FUNCTION_BLOCK FB_Servo
VAR_INPUT
	CAMTABLE		: MC_CAM_REF;
END_VAR
VAR_OUTPUT
END_VAR
VAR
	McPower: MC_Power;
	McReset: MC_Reset;
	McMoveAbs: MC_MoveAbsolute;
	McCamIN: MC_CamIn_V2;
	McCamOUT: MC_CamOut;
	McStop: MC_Stop;
	McWrite: MC_WriteMotionFunction;
	McRead: MC_ReadMotionFunction;
END_VAR
VAR_IN_OUT
	Axis			:	AXIS_REF;
	Slave			:	AXIS_REf;
	stAxisInterface	:	ST_AxisInterface;
END_VAR

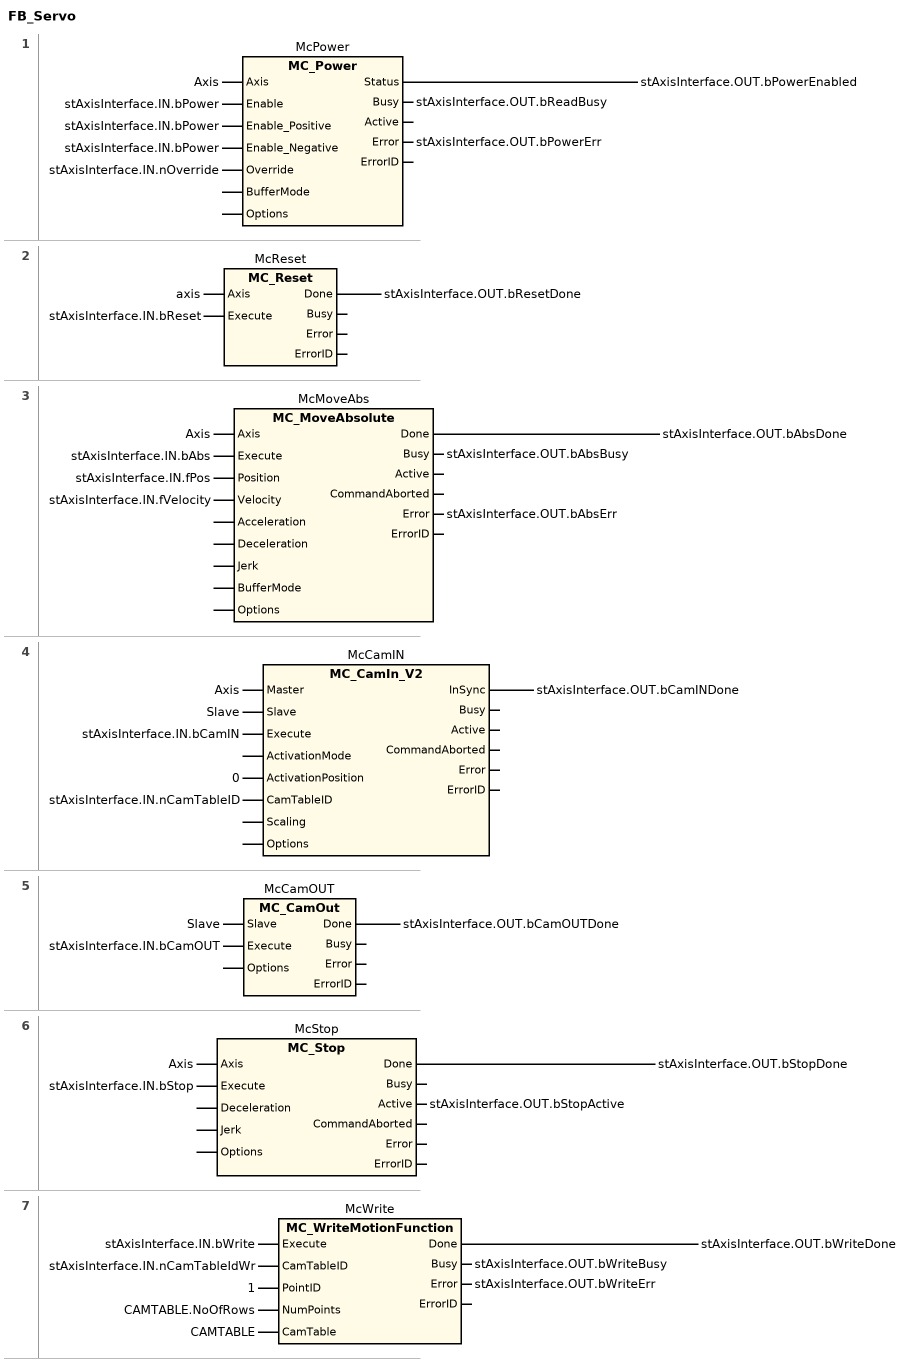
// NETWORK 1
McPower(
    Axis := Axis,
    Enable := stAxisInterface.IN.bPower,
    Enable_Positive := stAxisInterface.IN.bPower,
    Enable_Negative := stAxisInterface.IN.bPower,
    Override := stAxisInterface.IN.nOverride,
    Busy => stAxisInterface.OUT.bReadBusy,
    Error => stAxisInterface.OUT.bPowerErr); // MC_Power
stAxisInterface.OUT.bPowerEnabled := McPower.Status;

// NETWORK 2
McReset(Axis := axis, Execute := stAxisInterface.IN.bReset); // MC_Reset
stAxisInterface.OUT.bResetDone := McReset.Done;

// NETWORK 3
McMoveAbs(
    Axis := Axis,
    Execute := stAxisInterface.IN.bAbs,
    Position := stAxisInterface.IN.fPos,
    Velocity := stAxisInterface.IN.fVelocity,
    Busy => stAxisInterface.OUT.bAbsBusy,
    Error => stAxisInterface.OUT.bAbsErr); // MC_MoveAbsolute
stAxisInterface.OUT.bAbsDone := McMoveAbs.Done;

// NETWORK 4
McCamIN(
    Master := Axis,
    Slave := Slave,
    Execute := stAxisInterface.IN.bCamIN,
    ActivationPosition := 0,
    CamTableID := stAxisInterface.IN.nCamTableID); // MC_CamIn_V2
stAxisInterface.OUT.bCamINDone := McCamIN.InSync;

// NETWORK 5
McCamOUT(Slave := Slave, Execute := stAxisInterface.IN.bCamOUT); // MC_CamOut
stAxisInterface.OUT.bCamOUTDone := McCamOUT.Done;

// NETWORK 6
McStop(Axis := Axis, Execute := stAxisInterface.IN.bStop, Active => stAxisInterface.OUT.bStopActive); // MC_Stop
stAxisInterface.OUT.bStopDone := McStop.Done;

// NETWORK 7
McWrite(
    Execute := stAxisInterface.IN.bWrite,
    CamTableID := stAxisInterface.IN.nCamTableIdWr,
    PointID := 1,
    NumPoints := CAMTABLE.NoOfRows,
    CamTable := CAMTABLE,
    Busy => stAxisInterface.OUT.bWriteBusy,
    Error => stAxisInterface.OUT.bWriteErr); // MC_WriteMotionFunction
stAxisInterface.OUT.bWriteDone := McWrite.Done;

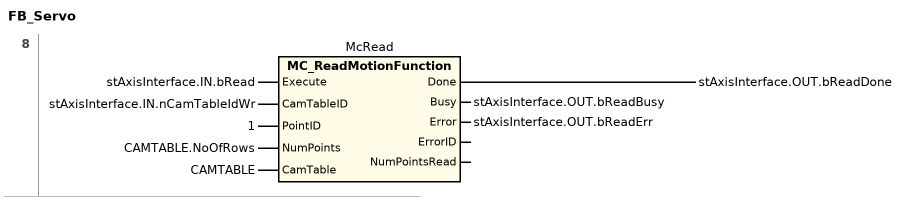
// NETWORK 8
McRead(
    Execute := stAxisInterface.IN.bRead,
    CamTableID := stAxisInterface.IN.nCamTableIdWr,
    PointID := 1,
    NumPoints := CAMTABLE.NoOfRows,
    CamTable := CAMTABLE,
    Busy => stAxisInterface.OUT.bReadBusy,
    Error => stAxisInterface.OUT.bReadErr); // MC_ReadMotionFunction
stAxisInterface.OUT.bReadDone := McRead.Done;

END_FUNCTION_BLOCK

(* stored: Version 1.1.0.1, ProductVersion 3.1.4022.18
   POU FB_Servo: Id {eed407d9-a361-4db5-9f96-5264fd2c7d6e}, SpecialFunc None *)
